// TwinCAT 3 PLC project testStepper
// ProgramVersion: 3.1.4023.0
// libraries:
//   Tc2_MC2, * (Beckhoff Automation GmbH)
//   Tc2_NC, * (Beckhoff Automation GmbH)
//   Tc2_Standard, * (Beckhoff Automation GmbH)
//   Tc2_System, * (Beckhoff Automation GmbH)
//   Tc3_Module, * (Beckhoff Automation GmbH)
//   VisuDialogs, * (System)
// project tree:
//   / GlobalTextList.TcGTLO (not stored), PlcTask.TcTTO (not stored), Visualization Manager.TcVMO (not stored)
//   GVLs/ GVL_AxisCtr.TcGVL (not stored), GVL_IO.TcGVL, GVL_NC.TcGVL (not stored)
//   POUs/ Command_to_Action.TcPOU, DegreesToRelativeMovment.TcPOU (not stored), movements.TcPOU (not stored), PositionToDegree.TcPOU, MAIN.TcPOU, POUNCPowerOn.TcPOU (not stored)
//   VISUs/ testStepperVisu.TcVIS (not stored)
// real-time tasks:
//   TASK PlcTask: cycle T#10ms, priority 20, ADS port 350
//   TASK PlcTask1: cycle T#10ms, priority 21, ADS port 351
// motion (NC):
//   TASK NC_test SAF: cycle T#2ms, priority 4, ADS port 501
//   TASK NC_test SVB: cycle T#10ms, priority 8, ADS port 511
//   AXIS Axis 1 (id 1)
//     OtherSettings: AllowMotionCmdToSlave=true
//     encoder EncType=1
//     drive DrvType=5
//       Analog: TorqueSetpointScale=10, ScaleFactorActTorque=0.1
//       TimeComp: TaskDelayCycles=1
//     controller CtrType=1
//       CtrPara: PriorControlFactor=1
//         Observer: BandWidth=20
// variable links:
//   testStepper/testStepper Instance <-> NC_test SAF/Axes/Axis 1
//     PlcTask Inputs/GVL_NC.stXAxis.NcToPlc <-> Outputs/ToPlc
//     PlcTask Outputs/GVL_NC.stXAxis.PlcToNc <-> Inputs/FromPlc

// ---- GVLs/GVL_IO.TcGVL
{attribute 'qualified_only'}
VAR_GLOBAL
	I_bXAxisLimitSwPos AT %I* : BOOL;
	I_bXAxisLimitSwNeg AT %I* : BOOL;
	
END_VAR

// ---- POUs/Command_to_Action.TcPOU
FUNCTION_BLOCK Command_to_Action
VAR_INPUT
	inputString : STRING;
END_VAR
VAR_OUTPUT
	recognitionValue : REAL;
END_VAR
VAR
	putString : STRING;
	recognitionString : STRING := 'Steer(';
	stringLength : int;
END_VAR

IF FIND(STR1:= inputString  , STR2:= recognitionString ) = 1 THEN
	putString := DELETE(STR:=inputString , LEN:= 6 , POS:=1 );
	stringLength := LEN(putstring);
	putString := DELETE(STR:=putString , LEN:= 1 , POS:= stringLength);
	recognitionValue := STRING_TO_INT(putString);
END_IF

END_FUNCTION_BLOCK

// ---- POUs/PositionToDegree.TcPOU
FUNCTION_BLOCK PositionToDegree
VAR_INPUT
	MaxPosition : LREAL;
	MaxSteeringAngle : INT;
	Position : LREAL;
END_VAR
VAR_OUTPUT
	Deg : LREAL;
END_VAR
VAR
END_VAR

IF (Position > 0 OR Position < 0) THEN
	Deg := (MaxSteeringAngle/MaxPosition)*Position;
ELSIF (Position = 0) THEN
	Deg := 0;		
END_IF

END_FUNCTION_BLOCK

// ---- POUs/MAIN.TcPOU
PROGRAM MAIN
VAR
	fbReadXaxisStatus: MC_ReadStatus;
	
END_VAR

fbReadXaxisStatus(
	Axis:=GVL_NC.stXAxis , 
	Enable:= GVL_AxisCtr.bXAxisEnable , 
	Valid=> , 
	Busy=> , 
	Error=> , 
	ErrorID=> , 
	ErrorStop=> , 
	Disabled=> , 
	Stopping=> , 
	StandStill=> , 
	DiscreteMotion=> , 
	ContinuousMotion=> , 
	SynchronizedMotion=> , 
	Homing=> , 
	ConstantVelocity=> , 
	Accelerating=> , 
	Decelerating=> , 
	Status=> GVL_NC.stXaxisStatus);
	POUNCPowerOn();
	movements();

END_PROGRAM
